TYPE EL5072_IND_InputsChannel :
STRUCT
	{attribute addProperty Name "Status"}
	Status AT %I* : EL5042_Status;
	{attribute addProperty Name "Position"}
	Position AT %I* : DINT;
	{attribute addProperty Name "Latch value"}
	LatchValue AT %I* : DINT;
END_STRUCT
END_TYPE

(* stored: Version 1.1.0.1, ProductVersion 3.1.4024.9
   DUT EL5072_IND_InputsChannel: Id {0f99de6b-165b-057a-1509-8dfe2a858674} *)
